// TIA Portal V20 export
// export: Created 2026-09-04T18:35:15.9542094Z, ExportSetting WithDefaults, DisplayName Totally Integrated Automation Portal, DisplayVersion V20, DisplayName TIA Portal Openness, DisplayVersion V20, DisplayName TIA Portal Version Control Interface, DisplayVersion V20, DisplayName STEP 7 Professional, DisplayVersion V20, DisplayName STEP 7 Safety, DisplayVersion V20, DisplayName WinCC Basic/Comfort/Advanced, DisplayVersion V20, DisplayName WinCC Professional, DisplayVersion V20, DisplayName WinCC Unified, DisplayVersion V20
DATA_BLOCK "Valve_Meta_DB"   // DB11
{ S7_Optimized_Access := 'TRUE' }
VERSION : 0.1
// stored: AutoNumber true, IsOnlyStoredInLoadMemory false, IsRetainMemResEnabled false, IsWriteProtectedInAS false, MemoryReserve 100
   VAR
      "Name" : Array[1..89] of String[20];
      Location : Array[1..89] of String[20];
      CmNo : Array[1..89] of String[6];
      VTag : Array[1..89] of String[12];
      SysName : Array[1..89] of String[12];
      FuncName : Array[1..89] of String[22];
      AftTblName : Array[1..14] of String[20];
      ErTblName : Array[1..14] of String[20];
      FwdTblName : Array[1..14] of String[20];
      AftTblLoc : Array[1..14] of String[20];
      ErTblLoc : Array[1..14] of String[20];
      FwdTblLoc : Array[1..14] of String[20];
      AftTblCmNo : Array[1..14] of String[6];
      ErTblCmNo : Array[1..14] of String[6];
      FwdTblCmNo : Array[1..14] of String[6];
      AftTblVTag : Array[1..14] of String[12];
      ErTblVTag : Array[1..14] of String[12];
      FwdTblVTag : Array[1..14] of String[12];
      AftTblFunc : Array[1..14] of String[22];
      ErTblFunc : Array[1..14] of String[22];
      FwdTblFunc : Array[1..14] of String[22];
      CfgTblName : Array[1..16] of String[20];
      CfgTblLoc : Array[1..16] of String[20];
      CfgTblCmNo : Array[1..16] of String[6];
      CfgTblVTag : Array[1..16] of String[12];
      CfgTblSys : Array[1..16] of String[12];
      CfgTblFunc : Array[1..16] of String[22];
      SelCmNo : String[6];
      SelVTag : String[12];
   END_VAR
BEGIN
   Location[1..2] := 'DB tank';
   Location[3] := 'Main line';
   Location[4] := 'Aft peak C';
   Location[5] := 'Aft peak';
   Location[6] := 'Aft peak P';
   Location[7] := 'Aft peak S';
   Location[8..13] := 'DB tank';
   Location[14..15] := 'Cross line';
   Location[16..17] := 'Pump 2';
   Location[18] := 'Main line';
   Location[19] := 'Pump 2';
   Location[20] := 'Pump 1';
   Location[21] := 'Bilge tie';
   Location[22] := 'Bilge system tie';
   Location[23..24] := 'Pump 2 discharge';
   Location[25] := 'Tank branch';
   Location[26] := 'Main line';
   Location[27] := 'Cross line';
   Location[28] := 'Bow thruster room';
   Location[29..30] := 'Hold 4';
   Location[31..32] := 'Hold 3';
   Location[33] := 'ER';
   Location[34] := 'ER/Pipe void';
   Location[35] := 'Pipe void aft';
   Location[36..37] := 'Engine Room';
   Location[38..39] := 'Hold 2';
   Location[40..41] := 'Hold 1';
   Location[42] := 'ER';
   Location[43] := 'Pump suction';
   Location[44] := 'ER';
   Location[45] := 'Void Deck';
   Location[46] := 'Pipe void aft';
   Location[47..48] := 'Hold 5';
   Location[49..50] := 'Discharge';
   Location[51] := 'Fire main';
   Location[52] := 'Fire line';
   Location[53] := 'Bilge Fire Pump 2';
   Location[54] := 'Bilge Fire Pump 1';
   Location[55] := 'TK6 High P';
   Location[56..57] := 'Manifold';
   Location[58] := 'TK5 Wing P';
   Location[59] := 'TK4 DB';
   Location[60] := 'Manifold';
   Location[61] := 'TK5 DB P';
   Location[62] := 'Manifold';
   Location[63] := 'TK3 Wing S';
   Location[64..66] := 'Manifold';
   Location[67] := 'TK2 Wing P';
   Location[68] := 'TK1 DB C';
   Location[69] := 'Main line';
   Location[70] := 'TK2 High C';
   Location[71] := 'Main line';
   Location[72] := 'TK2 Wing S';
   Location[73] := 'Fwd peak';
   Location[74] := 'Main line';
   Location[75] := 'Fwd peak';
   Location[76] := 'TK3 Wing P';
   Location[77..78] := 'Manifold';
   Location[79] := 'TK4 Wing P';
   Location[80] := 'TK4 Wing S';
   Location[81..82] := 'Manifold';
   Location[83] := 'TK3 DB';
   Location[84] := 'Cross line';
   Location[85..87] := 'Cross-over manifold';
   Location[89] := 'Cross-over manifold';
   CmNo[1] := 'CM25';
   CmNo[2] := 'CM26';
   CmNo[3] := 'CM50';
   CmNo[4] := 'CM51';
   CmNo[5] := 'CM52';
   CmNo[6] := 'CM53';
   CmNo[7] := 'CM54';
   CmNo[8] := 'CM55';
   CmNo[9] := 'CM56';
   CmNo[10] := 'CM57';
   CmNo[11] := 'CM58';
   CmNo[12] := 'CM59';
   CmNo[13] := 'CM60';
   CmNo[14] := 'CM67';
   CmNo[15] := 'CM68';
   CmNo[16] := 'CM69';
   CmNo[17] := 'CM70';
   CmNo[18] := 'CM71';
   CmNo[19] := 'CM72';
   CmNo[20] := 'CM78';
   CmNo[21] := 'CM79';
   CmNo[22] := 'CM80';
   CmNo[23] := 'CM81';
   CmNo[24] := 'CM82';
   CmNo[25] := 'CM83';
   CmNo[26] := 'CM84';
   CmNo[27] := 'CM85';
   CmNo[28] := 'CM01';
   CmNo[29] := 'CM02';
   CmNo[30] := 'CM03';
   CmNo[31] := 'CM04';
   CmNo[32] := 'CM05';
   CmNo[33] := 'CM06';
   CmNo[34] := 'CM07';
   CmNo[35] := 'CM08';
   CmNo[36] := 'CM09';
   CmNo[37] := 'CM10';
   CmNo[38] := 'CM11';
   CmNo[39] := 'CM12';
   CmNo[40] := 'CM13';
   CmNo[41] := 'CM14';
   CmNo[42] := 'CM15';
   CmNo[43] := 'CM16';
   CmNo[44] := 'CM17';
   CmNo[45] := 'CM18';
   CmNo[46] := 'CM19';
   CmNo[47] := 'CM20';
   CmNo[48] := 'CM21';
   CmNo[49] := 'CM23';
   CmNo[50] := 'CM24';
   CmNo[51] := 'CM94';
   CmNo[52] := 'CM95';
   CmNo[53] := 'CM96';
   CmNo[54] := 'CM97';
   CmNo[55] := 'CM27';
   CmNo[56] := 'CM28';
   CmNo[57] := 'CM29';
   CmNo[58] := 'CM30';
   CmNo[59] := 'CM31';
   CmNo[60] := 'CM32';
   CmNo[61] := 'CM33';
   CmNo[62] := 'CM34';
   CmNo[63] := 'CM35';
   CmNo[64] := 'CM36';
   CmNo[65] := 'CM37';
   CmNo[66] := 'CM38';
   CmNo[67] := 'CM39';
   CmNo[68] := 'CM40';
   CmNo[69] := 'CM41';
   CmNo[70] := 'CM42';
   CmNo[71] := 'CM43';
   CmNo[72] := 'CM44';
   CmNo[73] := 'CM45';
   CmNo[74] := 'CM46';
   CmNo[75] := 'CM47';
   CmNo[76] := 'CM48';
   CmNo[77] := 'CM49';
   CmNo[78] := 'CM61';
   CmNo[79] := 'CM62';
   CmNo[80] := 'CM63';
   CmNo[81] := 'CM64';
   CmNo[82] := 'CM65';
   CmNo[83] := 'CM66';
   CmNo[84] := 'CM77';
   CmNo[85] := 'CM86';
   CmNo[86] := 'CM87';
   CmNo[87] := 'CM88';
   CmNo[88] := 'CM89';
   CmNo[89] := 'CM90';
   VTag[1] := '11-020-A1';
   VTag[2] := '11-021-A1';
   VTag[3] := '11-008-A1';
   VTag[4] := '11-009-A1';
   VTag[5] := '11-010-A1';
   VTag[6] := '11-060-A1';
   VTag[7] := '11-061-A1';
   VTag[8] := '11-024-A2';
   VTag[9] := '11-025-A2';
   VTag[10] := '11-028-A1';
   VTag[11] := '11-029-A1';
   VTag[12] := '11-022-A2';
   VTag[13] := '11-023-A2';
   VTag[14] := '11-001-A2';
   VTag[15] := '11-004-A1';
   VTag[16] := '11-002-A2';
   VTag[17] := '11-002-A4';
   VTag[18] := '11-005-A1';
   VTag[19] := '11-006-A1';
   VTag[20] := '11-011-A1';
   VTag[21] := '11-011-A3';
   VTag[22] := '11-011-A4';
   VTag[23] := '11-012-A1';
   VTag[24] := '11-012-A3';
   VTag[25] := '11-015-A1';
   VTag[26] := '11-016-A1';
   VTag[27] := '11-003-A1';
   VTag[28] := '10-041-A1';
   VTag[29] := '10-017-A1';
   VTag[30] := '10-018-A1';
   VTag[31] := '10-021-A1';
   VTag[32] := '10-022-A1';
   VTag[33] := '10-007-A1';
   VTag[34] := '10-009-A1';
   VTag[35] := '10-012-A1';
   VTag[36] := '10-001-A1';
   VTag[37] := '10-002-A1';
   VTag[38] := '10-025-A1';
   VTag[39] := '10-026-A1';
   VTag[40] := '10-034-A1';
   VTag[41] := '10-035-A1';
   VTag[42] := '10-003-A1';
   VTag[43] := '10-004-A1';
   VTag[44] := '10-005-A1';
   VTag[45] := '10-001-A2';
   VTag[46] := '10-013-A1';
   VTag[47] := '10-010-A1';
   VTag[48] := '10-011-A1';
   VTag[49] := '10-046-A1';
   VTag[50] := '10-047-A2';
   VTag[51] := '20-023-A1';
   VTag[52] := '20-025-A1';
   VTag[53] := '20-022-A1';
   VTag[54] := '20-024-A1';
   VTag[55] := '11-030-A1';
   VTag[56] := '11-031-A1';
   VTag[57] := '11-032-A1';
   VTag[58] := '11-033-A1';
   VTag[59] := '11-034-A2';
   VTag[60] := '11-035-A1';
   VTag[61] := '11-036-A1';
   VTag[62] := '11-037-A1';
   VTag[63] := '11-046-A1';
   VTag[64] := '11-047-A2';
   VTag[65] := '11-048-A1';
   VTag[66] := '11-049-A1';
   VTag[67] := '11-050-A1';
   VTag[68] := '11-051-A1';
   VTag[69] := '11-052-A1';
   VTag[70] := '11-053-A1';
   VTag[71] := '11-054-A2';
   VTag[72] := '11-055-A1';
   VTag[73] := '11-056-A1';
   VTag[74] := '11-057-A1';
   VTag[75] := '11-058-A1';
   VTag[76] := '11-042-A1';
   VTag[77] := '11-043-A1';
   VTag[78] := '11-043-A2';
   VTag[79] := '11-041-A2';
   VTag[80] := '11-039-A1';
   VTag[81] := '11-040-A1';
   VTag[82] := '11-044-A2';
   VTag[83] := '11-045-A2';
   VTag[84] := '11-014-A1';
   VTag[85] := '11-063-A1';
   VTag[86] := '11-064-A1';
   VTag[87] := '11-065-A1';
   VTag[88] := '11-066-A1';
   VTag[89] := '11-067-A1';
   SysName[1..27] := 'Ballast Aft';
   SysName[28..54] := 'Bilge';
   SysName[55..89] := 'Ballast Fwd';
   FuncName[1] := 'Filling';
   FuncName[2] := 'Suction';
   FuncName[3..5] := 'Isolation';
   FuncName[6..7] := 'Tank suction';
   FuncName[8] := 'Filling';
   FuncName[9..10] := 'Suction';
   FuncName[11] := 'Filling';
   FuncName[12] := 'Suction';
   FuncName[13] := 'Filling';
   FuncName[14..17] := 'Isolation';
   FuncName[18] := 'Distribution';
   FuncName[19] := 'Suction';
   FuncName[20] := 'Discharge';
   FuncName[21] := 'Cross connect';
   FuncName[22..27] := 'Isolation';
   FuncName[28..32] := 'Bilge suction';
   FuncName[33] := 'Suction';
   FuncName[34..35] := 'Isolation';
   FuncName[36] := 'Suction';
   FuncName[37] := 'Main suction';
   FuncName[38..41] := 'Bilge suction';
   FuncName[42] := 'Suction';
   FuncName[43] := 'Isolation';
   FuncName[44] := 'Suction';
   FuncName[45] := 'Bilge suction';
   FuncName[46] := 'Isolation';
   FuncName[47..48] := 'Bilge suction';
   FuncName[49..51] := 'Isolation';
   FuncName[52] := 'Fire/Bilge crossover';
   FuncName[53..54] := 'Seawater priming';
   FuncName[55] := 'Filling';
   FuncName[56..57] := 'Suction';
   FuncName[58..59] := 'Filling';
   FuncName[60] := 'Suction';
   FuncName[61] := 'Filling';
   FuncName[62] := 'Suction';
   FuncName[63] := 'Filling';
   FuncName[64..66] := 'Suction';
   FuncName[67..68] := 'Filling';
   FuncName[69] := 'Isolation';
   FuncName[70] := 'Filling';
   FuncName[71] := 'Isolation';
   FuncName[72..73] := 'Filling';
   FuncName[74] := 'Isolation';
   FuncName[75..76] := 'Filling';
   FuncName[77..78] := 'Suction';
   FuncName[79..80] := 'Filling';
   FuncName[81..82] := 'Suction';
   FuncName[83] := 'Filling';
   FuncName[84..87] := 'Isolation';
   FuncName[89] := 'Isolation';
END_DATA_BLOCK
